FUNCTION_BLOCK novobloc (* oi *)
  (* Standard: 61499-2 *)
  (* Version 11-01-12, GASR *)
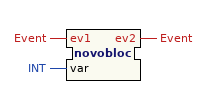
  EVENT_INPUT
    ev1;
  END_EVENT
  EVENT_OUTPUT
    ev2;
  END_EVENT
  VAR_INPUT
    var : INT;
  END_VAR
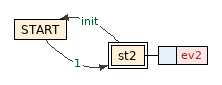
  EC_STATES
    st2 : -> ev2;
    START;
  END_STATES
  EC_TRANSITIONS
    st2 TO START := init;
    START TO st2 := 1;
  END_TRANSITIONS
END_FUNCTION_BLOCK
